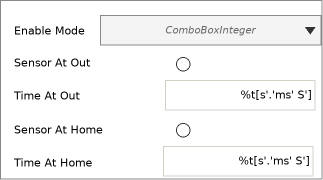
VISUALIZATION visStandardCylinderSettings  // 323x180
VAR_INPUT
	refSetting : REFERENCE TO ST_StandardCylinderSettings;
END_VAR
VAR CONSTANT
	cMinTime : DINT := 0;
	cMaxTime : DINT := T#100S;
	sDialog1 : STRING := 'Time at out';
	sDialog2 : STRING := 'Time at home';
END_VAR
    Label (11,48 150x30), "Sensor At Out"
    Label (11,81 150x30), "Time At Out"
    Label (11,148 150x30), "Time At Home"
    Label (11,115 150x30), "Sensor At Home"
    RadioButton (174,49 132x30), variable: refSetting.bSensorAtOut
        Areas[0]: Text=Off
        Areas[1]: Text=On
    Label (11,16 150x30), "Enable Mode"
    ComboBoxInteger (100,15 221x30), variable: refSetting.eEnableMode, text list: 'txtLstCylinderEnableMode'
    RadioButton (174,115 132x30), variable: refSetting.bSensorAtHome
        Areas[0]: Text=Off
        Areas[1]: Text=On
    Textfield (163,146 150x30), "%t[s'.'ms' S']", text variable: refSetting.tTimeToOrAtHome
        OnMouseClick: write the text variable via Default, min cMinTime, max cMaxTime, title sDialog2
    Textfield (165,80 150x30), "%t[s'.'ms' S']", text variable: refSetting.tTimeToOrAtOut
        OnMouseClick: write the text variable via Default, min cMinTime, max cMaxTime, title sDialog1
END_VISUALIZATION

(* stored: Version 1.1.0.1, ProductVersion 3.1.4019.2
   Visu visStandardCylinderSettings: Id {d3160ccb-7dbe-484b-9732-04c64e22535d} *)
